TYPE ST_Point :
STRUCT
	x	: LREAL;
	y	: LREAL;	
END_STRUCT
END_TYPE

(* stored: Version 1.1.0.1, ProductVersion 3.1.4024.9
   DUT ST_Point: Id {1200598e-9cda-4a42-a8ab-ac3203af9fc9} *)
